(* PLC project Tc2_Utilities.FB_LicFileCopyToDongle Demo, tc3-libraries-kb TwinCAT 3.1 *)
(* stored: creationDateTime 2026-05-10T20:00:00, modificationDateTime 2026-05-10T20:00:00 *)

PROGRAM P_Demo_FB_LicFileCopyToDongle
  VAR
    fbFB_LicFileCopyToDongle : FB_LicFileCopyToDongle;  (* Tc2_Utilities.FB_LicFileCopyToDongle 实例 *)
    arg_sNetIdSrc : T_AmsNetId;  (* VAR_INPUT sNetIdSrc *)
    arg_sNetIdDest : T_AmsNetId;  (* VAR_INPUT sNetIdDest *)
    arg_nPortDest : UINT;  (* VAR_INPUT nPortDest *)
    arg_sFilePathNameSrc : T_MaxString;  (* VAR_INPUT sFilePathNameSrc *)
    arg_sFileNameDest : STRING;  (* VAR_INPUT sFileNameDest *)
    arg_pCopyBuff : PVOID;  (* VAR_INPUT pCopyBuff *)
    arg_cbCopyLen : UDINT;  (* VAR_INPUT cbCopyLen *)
    arg_bExecute : BOOL;  (* VAR_INPUT bExecute *)
    arg_dwPassCode : DWORD;  (* VAR_INPUT dwPassCode *)
    arg_tTimeout : TIME;  (* VAR_INPUT tTimeout *)
    out_bBusy : BOOL;  (* VAR_OUTPUT bBusy *)
    out_bError : BOOL;  (* VAR_OUTPUT bError *)
    out_nErrorId : UDINT;  (* VAR_OUTPUT nErrorId *)
  END_VAR

            // ============================================================
// Tc2_Utilities.FB_LicFileCopyToDongle 演示程序（FB 实例）
// ============================================================
// 验证步骤：
//   1. 引用 Tc2_Utilities（及依赖类型所在库 Tc2_System 等）
//   2. 编译 + 登录
//   3. 按 doc.md 给 arg_* 赋值
//   4. 在线监视 out_* / io_* 输出
// ============================================================

fbFB_LicFileCopyToDongle(
    sNetIdSrc := arg_sNetIdSrc,
    sNetIdDest := arg_sNetIdDest,
    nPortDest := arg_nPortDest,
    sFilePathNameSrc := arg_sFilePathNameSrc,
    sFileNameDest := arg_sFileNameDest,
    pCopyBuff := arg_pCopyBuff,
    cbCopyLen := arg_cbCopyLen,
    bExecute := arg_bExecute,
    dwPassCode := arg_dwPassCode,
    tTimeout := arg_tTimeout,
    bBusy => out_bBusy,
    bError => out_bError,
    nErrorId => out_nErrorId
);

          
END_PROGRAM
